Staubli VAL3: Control_Bottom.pgx

public program Control_Bottom(string& x_sBottomList[])
  local num l_nIndex
  local num l_nNum
begin
  //说明：
  //函数功能：对功能键进行说明
  //x_sBottomList 功能键说明，通过字符串数组来实现


  //参数初始化
  setTextMode(0)
  l_nNum=min(7,size(x_sBottomList)-1)


  for l_nIndex=0 to  l_nNum
    gotoxy(1+l_nIndex*5,13)
    put(left(x_sBottomList[l_nIndex]+"       ",4+len(x_sBottomList[l_nIndex])-getDisplayLen(x_sBottomList[l_nIndex])))
  endFor

  //补全
  if l_nNum<7
    for l_nIndex=l_nNum to 7
      gotoxy(1+l_nIndex*5,13)
      put("  ")
    endFor
  endIf
end
